{attribute 'qualified_only'}
VAR_GLOBAL
	Robot1	:	TcoMitsubishiRobotics.TcoCr800_IO_v_1_x_x;
END_VAR

(* stored: Version 1.1.0.1, ProductVersion 3.1.4024.12
   GVL GVL: Id {48a67708-8b9b-0e10-0989-f4d99d2933ce} *)
